TYPE TempIn :
STRUCT
     (****INPUT**)
   iPV:                                  INT;// 读取当前温度 (模块) 
   fPV:                                  REAL;// 读取当前温度(转换后)



  (****Status**)
   SaveParaOK:                      BOOL;           //保存参数OK
   PIDON:                             BOOL;          //PID功能开启
   AutoTuningON:                  BOOL;          //自整定开启
   AutoTuningerr:                   BOOL;          //自整定故障
   HeatingON:                       BOOL;          //加热中
   CoolingON:                       BOOL;          //制冷中
   AutoTuningOK:                  BOOL;          //自整定OK

END_STRUCT
END_TYPE

(* stored: Version 1.1.0.1, ProductVersion 3.1.4024.9
   DUT TempIn: Id {9cd403a9-1ebb-476a-a171-d724b3989ad4} *)
